PROGRAM Reel
VAR
	Zero: MC_SetPosition;
	power: MC_Power;
	MC_MoveAbsolute: MC_MoveAbsolute;
END_VAR

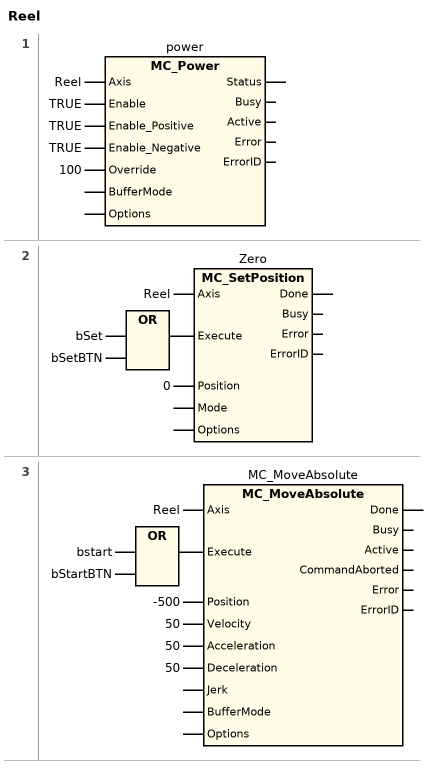
// NETWORK 1
power(Axis := Reel, Enable := TRUE, Enable_Positive := TRUE, Enable_Negative := TRUE, Override := 100); // MC_Power

// NETWORK 2
Zero(Axis := Reel, Execute := bSet OR bSetBTN, Position := 0); // MC_SetPosition

// NETWORK 3
MC_MoveAbsolute(
    Axis := Reel,
    Execute := bstart OR bStartBTN,
    Position := -500,
    Velocity := 50,
    Acceleration := 50,
    Deceleration := 50);

END_PROGRAM

(* stored: Version 1.1.0.1, ProductVersion 3.1.4024.12
   POU Reel: Id {d557e279-5996-4de8-b528-0b9d0286dce8}, SpecialFunc None *)
